{attribute 'GeneratedUsingTerminal: ELX3252-0000-0016'}
{attribute addProperty BoxType "ELX3252-0000-0016"}
{attribute addProperty Id "EtcSlaveTerminalBaseAI_Standard_Channel_1AT %I*AI_Standard_Channel_3D09D60D7AI_Standard_Channel_2AT %I*AI_Standard_Channel_3D09D60D7WcStateAT %I*WcState_9091E0EB2InfoDataAT %I*InfoData_32EB74EA10"}
{attribute addProperty CRC "2120444076"}
{attribute addProperty Size "26"}
TYPE ELX3252_7E6368AC EXTENDS EtcSlaveTerminalBase :
STRUCT
	{attribute addProperty Name "AI_Standard_Channel_1"}
	AI_Standard_Channel_1 : AI_Standard_Channel_3D09D60D;
	{attribute addProperty Name "AI_Standard_Channel_2"}
	AI_Standard_Channel_2 : AI_Standard_Channel_3D09D60D;
	{attribute addProperty Name "WcState"}
	WcState : WcState_9091E0EB;
	{attribute addProperty Name "InfoData"}
	InfoData : InfoData_32EB74EA;
END_STRUCT
END_TYPE

(* stored: Version 1.2.0.0, ProductVersion 3.1.4024.9
   DUT ELX3252_7E6368AC: Id {4fc5ccbe-b14a-41f2-87ab-487850e929f9} *)
